FUNCTION_BLOCK ConveyorControllerISub (* Conveyor Controller Interface subscribe *)
  (* Standard: 61499-2 *)
  (* Version 0.2, 2003-12-05, JHC, Rockwell Automation, Renamed from NEWCOMPFB. *)
  (* Version 0.1, 2002-01-08, JHC, Rockwell Automation, Added DLY FB as example. *)
  (* Version 0.0, 2000-05-27, JHC, Rockwell Automation *)
  (* Compiler header: package fb.rt.dasdA1.A2.Conveyor; *)
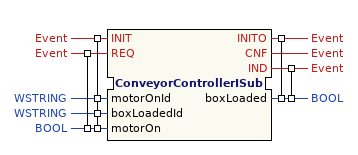
  EVENT_INPUT
    INIT WITH motorOnId, boxLoadedId, motorOn; (* Initialization Request *)
    REQ WITH motorOn; (* Normal Execution Request *)
  END_EVENT
  EVENT_OUTPUT
    INITO WITH boxLoaded; (* Initialization Confirm *)
    CNF; (* Execution Confirmation *)
    IND WITH boxLoaded;
  END_EVENT
  VAR_INPUT
    motorOnId : WSTRING;
    boxLoadedId : WSTRING;
    motorOn : BOOL;
  END_VAR
  VAR_OUTPUT
    boxLoaded : BOOL;
  END_VAR
  FBS
    pusherColorSensor : SUBL_1;
    pusherPush : PUBL_1;
  END_FBS
  EVENT_CONNECTIONS
    pusherColorSensor.INITO TO INITO;
    pusherColorSensor.IND TO CNF;
    INIT TO pusherPush.INIT;
    REQ TO pusherPush.REQ;
    pusherPush.INITO TO pusherColorSensor.INIT;
    pusherPush.CNF TO CNF;
    pusherColorSensor.IND TO IND;
  END_CONNECTIONS
  DATA_CONNECTIONS
    boxLoadedId TO pusherColorSensor.ID;
    pusherColorSensor.RD_1 TO boxLoaded;
    motorOn TO pusherPush.SD_1;
    motorOnId TO pusherPush.ID;
  END_CONNECTIONS
END_FUNCTION_BLOCK
